(* Schneider Machine Expert - Basic project Pump_Tank_TM221, file version 3.0.0.0 *)
(* ProjectInformations: Name=New project *)

HARDWARE
  Cpu 0: TM221CE24T
  EthernetConfiguration: NetworkName=M221, IpAllocationMode=FixedAddress, IpAddress=0.0.0.0, SubnetMask=0.0.0.0
  SerialLineConfiguration: Baud=Baud19200, Parity=ParityEven, DataBits=DataBits8, StopBits=StopBits1, PhysicalMedium=PhysicalMediumRs485, TransmissionMode=TransmissionModeModbusRtu, SlaveId=1, Addressing=SlaveAddressing
  MastTask: UsePeriodScanMode=false, PeriodScan=100
  FastTask: Period=255
  CpuBehavior: StartingMode=StartAsPreviousState, AutoSaveRamOnEeprom=true, WatchdogPeriod=250

SYMBOLS  (address, symbol, comment, settings)
  %TM0      PUMP1_DELAY  "Pump 1 Startup Delay 2s"  [Type=TON, TimeBase=TimeBase1s, Preset=2]
  %TM1      PUMP2_DELAY  "Pump 2 Startup Delay 2s"  [Type=TON, TimeBase=TimeBase1s, Preset=2]
  %TM2      PUMP3_DELAY  "Pump 3 Startup Delay 2s"  [Type=TON, TimeBase=TimeBase1s, Preset=2]
  %I0.0     START_BTN
  %I0.1     STOP_BTN
  %I0.2     EMERGENCY
  %Q0.0     LIGHT_1
  %Q0.2     LIGHT_3

POU Pump_Tank_Main
  (* SectionNumber=1 *)

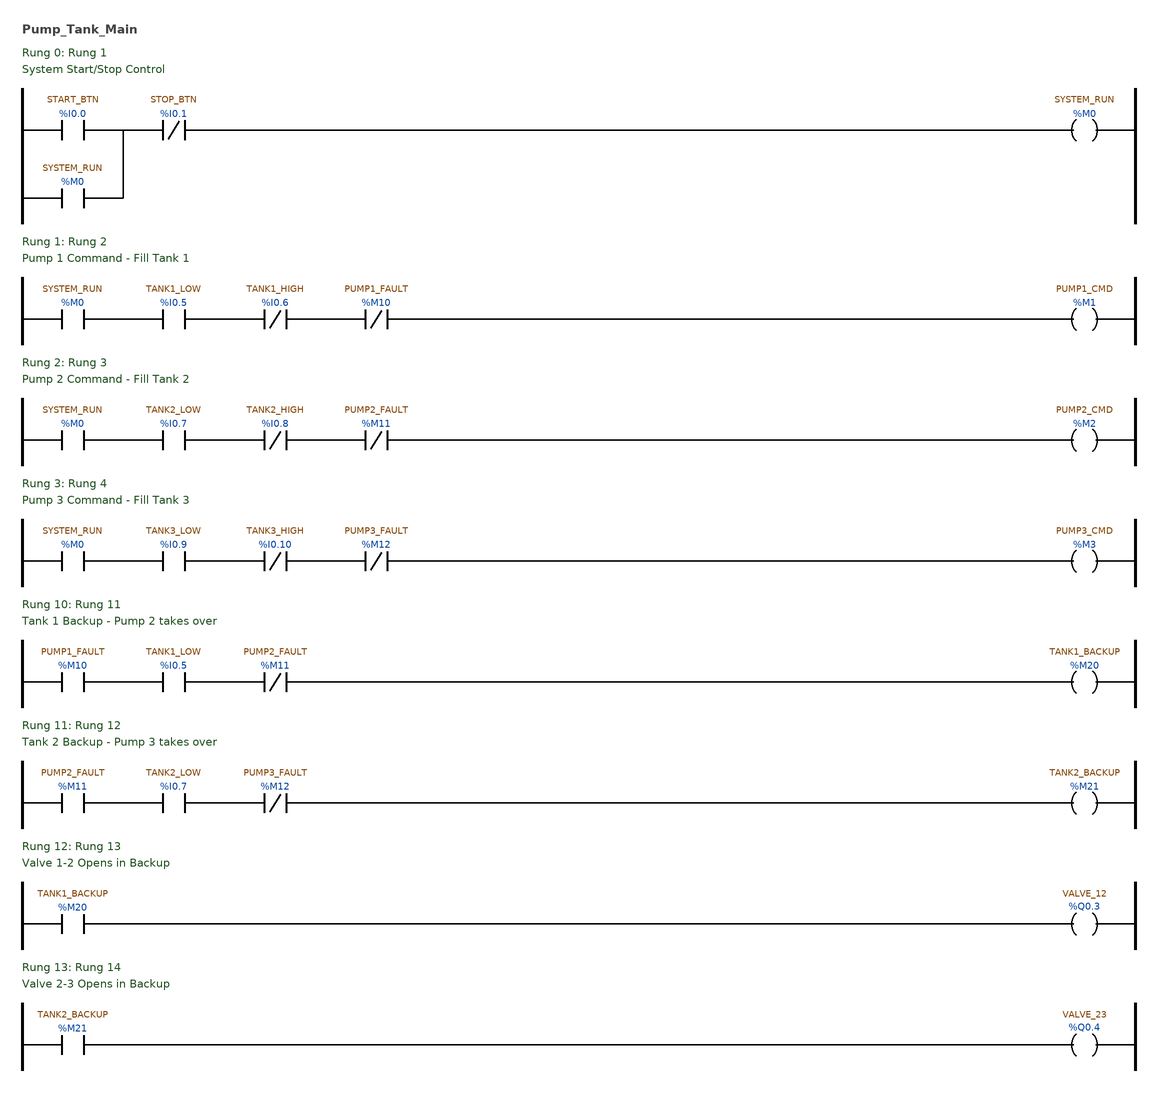

// Rung 0: Rung 1
// System Start/Stop Control
  LD %I0.0                (* START_BTN - Load START *)
  OR %M0                  (* Seal-in *)
  ANDN %I0.1              (* STOP_BTN - AND NOT STOP *)
  ST %M0                  (* SYSTEM_RUN *)
  // %I0.0: Start Button
  // %M0: Seal-in
  // %I0.1: Stop Button NC
  // %M0: System Running
  // as ST:
  //   %M0 := (START_BTN OR %M0) AND NOT STOP_BTN;

// Rung 1: Rung 2
// Pump 1 Command - Fill Tank 1
  LD %M0
  AND %I0.5               (* Tank 1 low *)
  ANDN %I0.6              (* Not high *)
  ANDN %M10               (* No fault *)
  ST %M1
  // as ST:
  //   %M1 := %M0 AND %I0.5 AND NOT %I0.6 AND NOT %M10;

// Rung 2: Rung 3
// Pump 2 Command - Fill Tank 2
  LD %M0
  AND %I0.7
  ANDN %I0.8
  ANDN %M11
  ST %M2
  // as ST:
  //   %M2 := %M0 AND %I0.7 AND NOT %I0.8 AND NOT %M11;

// Rung 3: Rung 4
// Pump 3 Command - Fill Tank 3
  LD %M0
  AND %I0.9
  ANDN %I0.10
  ANDN %M12
  ST %M3
  // as ST:
  //   %M3 := %M0 AND %I0.9 AND NOT %I0.10 AND NOT %M12;

// Rung 4: Rung 5
// Pump 1 Timer + Output
  BLK %TM0                (* PUMP1_DELAY *)
  LD %M1
  IN
  END_BLK
  LD %M1
  ST %Q0.0                (* LIGHT_1 *)
  // as ST:
  //   PUMP1_DELAY(IN := %M1);
  //   LIGHT_1 := %M1;
  (* the ladder stored for this rung does not match its IL; not drawn *)

// Rung 5: Rung 6
// Pump 1 Zero Speed Fault - Latching
  LD %TM0.Q               (* PUMP1_DELAY - Timer done *)
  ANDN %I0.2              (* EMERGENCY - No speed *)
  OR %M10                 (* Latch *)
  ANDN %I0.11             (* Not reset *)
  ST %M10
  // as ST:
  //   %M10 := (PUMP1_DELAY.Q AND NOT EMERGENCY OR %M10) AND NOT %I0.11;
  (* the ladder stored for this rung does not match its IL; not drawn *)

// Rung 6: Rung 7
// Pump 2 Output + Backup for Tank 1
  LD %M2
  OR %M20                 (* Backup Tank1 *)
  ST %Q0.1
  // as ST:
  //   %Q0.1 := %M2 OR %M20;
  (* the ladder stored for this rung does not match its IL; not drawn *)

// Rung 7: Rung 8
// Pump 2 Zero Speed Fault
  LD %TM1.Q               (* PUMP2_DELAY *)
  ANDN %I0.3
  OR %M11
  ANDN %I0.11
  ST %M11
  // as ST:
  //   %M11 := (PUMP2_DELAY.Q AND NOT %I0.3 OR %M11) AND NOT %I0.11;
  (* the ladder stored for this rung does not match its IL; not drawn *)

// Rung 8: Rung 9
// Pump 3 Output + Backup for Tank 2
  LD %M3
  OR %M21
  ST %Q0.2                (* LIGHT_3 *)
  // as ST:
  //   LIGHT_3 := %M3 OR %M21;
  (* the ladder stored for this rung does not match its IL; not drawn *)

// Rung 9: Rung 10
// Pump 3 Zero Speed Fault
  LD %TM2.Q               (* PUMP3_DELAY *)
  ANDN %I0.4
  OR %M12
  ANDN %I0.11
  ST %M12
  // as ST:
  //   %M12 := (PUMP3_DELAY.Q AND NOT %I0.4 OR %M12) AND NOT %I0.11;
  (* the ladder stored for this rung does not match its IL; not drawn *)

// Rung 10: Rung 11
// Tank 1 Backup - Pump 2 takes over
  LD %M10
  AND %I0.5
  ANDN %M11
  ST %M20
  // as ST:
  //   %M20 := %M10 AND %I0.5 AND NOT %M11;

// Rung 11: Rung 12
// Tank 2 Backup - Pump 3 takes over
  LD %M11
  AND %I0.7
  ANDN %M12
  ST %M21
  // as ST:
  //   %M21 := %M11 AND %I0.7 AND NOT %M12;

// Rung 12: Rung 13
// Valve 1-2 Opens in Backup
  LD %M20
  ST %Q0.3
  // as ST:
  //   %Q0.3 := %M20;

// Rung 13: Rung 14
// Valve 2-3 Opens in Backup
  LD %M21
  ST %Q0.4
  // as ST:
  //   %Q0.4 := %M21;

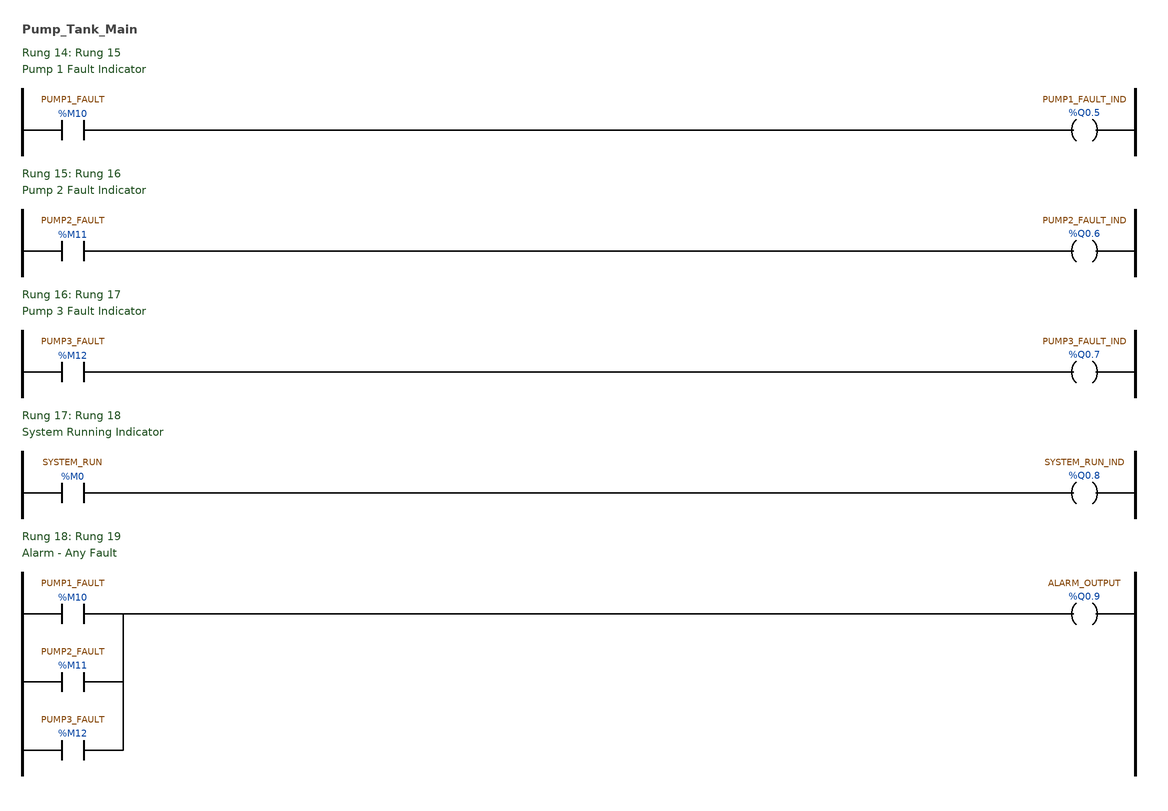

// Rung 14: Rung 15
// Pump 1 Fault Indicator
  LD %M10
  ST %Q0.5
  // as ST:
  //   %Q0.5 := %M10;

// Rung 15: Rung 16
// Pump 2 Fault Indicator
  LD %M11
  ST %Q0.6
  // as ST:
  //   %Q0.6 := %M11;

// Rung 16: Rung 17
// Pump 3 Fault Indicator
  LD %M12
  ST %Q0.7
  // as ST:
  //   %Q0.7 := %M12;

// Rung 17: Rung 18
// System Running Indicator
  LD %M0
  ST %Q0.8
  // as ST:
  //   %Q0.8 := %M0;

// Rung 18: Rung 19
// Alarm - Any Fault
  LD %M10
  OR %M11
  OR %M12
  ST %Q0.9
  // as ST:
  //   %Q0.9 := %M10 OR %M11 OR %M12;
